(* IEC 61131-3 sources: volt/packages/volt-lsp-iec/test-corpus/lenze-mid/Device/Plc Logic/Application/Library Manager/CDSV3ProtocolUtils, 39 files *)

(* ---- PROTOCOLDATAUNIT.dut ---- *)
TYPE PROTOCOLDATAUNIT :
STRUCT
	PDATA : POINTER TO BYTE;
	DWSIZE : DWORD;
END_STRUCT
END_TYPE

(* ---- SERVICEHEADER.dut ---- *)
TYPE SERVICEHEADER :
STRUCT
	HEADERTAG : UINT := Constants.HeaderTagStandard;
	HEADERSIZE : UINT := UDINT_TO_UINT((SIZEOF(THIS^) - 4));
	SERVICEGROUP : UINT;
	SERVICE : UINT;
	DEVICESESSIONID : UDINT;
	SERVICELENGTH : UDINT;
	CUSTOMERID : UINT := 0;
	RESERVED : UINT := 0;
END_STRUCT
END_TYPE

(* ---- CONSTANTS.gvl ---- *)
VAR_GLOBAL
	HEADERTAGSTANDARD : UINT := 16#CD55;
	TAG_GENERALERROR : UINT := 16#FF7F;
	TAG_EXTENDEDERRORINFO : UINT := 16#FF7E;
END_VAR

(* ---- ERRORS.gvl ---- *)
VAR_GLOBAL
	ERR_PLCS_UNKNOWN_PROTOCOL : UDINT := 16#1011;
	ERR_PLCS_ALIGNMENT : UDINT := 16#1010;
	ERR_TSW_NOTCREATED : UDINT := 16#1000;
	ERR_TSR_NOMORETAGS : UDINT := 16#1040;
	ERR_TSR_NOCONTAINERTAG : UDINT := 16#1041;
	ERR_TSR_NODATATAG : UDINT := 16#1042;
	ERR_TSR_ENDOFTAG : UDINT := 16#1043;
	ERR_TSR_READONWRONGTAG : UDINT := 16#1044;
	ERR_TSR_NOTCREATED : UDINT := 16#1045;
END_VAR

(* ---- ICDSV3REQUESTBUILDER.itf ---- *)
INTERFACE ICDSV3REQUESTBUILDER
END_INTERFACE

METHOD BUILDREQUEST : UDINT
VAR_INPUT
	ITFSERVICEWRITER : IServiceWriter;
	XHASTOSWAP : BOOL;
END_VAR
END_METHOD

METHOD GETDATABUFFER : POINTER TO BYTE
END_METHOD

METHOD GETDATABUFFERSIZE : UDINT
END_METHOD

METHOD GETSERVICE : UINT
END_METHOD

METHOD GETSERVICEGROUP : UINT
END_METHOD

METHOD REQUESTENQUEUED : UDINT
END_METHOD

(* ---- ICDSV3REQUESTCALLBACK.itf ---- *)
INTERFACE ICDSV3REQUESTCALLBACK
END_INTERFACE

METHOD SETTARGETBYTEORDER
VAR_INPUT
	EBYTEORDER : IDatasources.ByteOrder;
END_VAR
END_METHOD

(* ---- IREQUESTRESULT.itf ---- *)
INTERFACE IREQUESTRESULT
END_INTERFACE

METHOD ISREPLYPENDING : BOOL
END_METHOD

METHOD SETREPLYPENDING
VAR_INPUT
	XREPLYPENDING : BOOL;
END_VAR
END_METHOD

(* ---- ISERVICEREADER.itf ---- *)
INTERFACE ISERVICEREADER
END_INTERFACE

METHOD GETCONTENT : UDINT
VAR_OUTPUT
	PDATA : POINTER TO BYTE;
END_VAR
END_METHOD

METHOD GETCONTENTSIZE : UDINT
VAR_OUTPUT
	CONTENTSIZE : UDINT;
END_VAR
END_METHOD

METHOD GETUNREADCONTENT : UDINT
VAR_OUTPUT
	PDATA : POINTER TO BYTE;
END_VAR
END_METHOD

METHOD GETUNREADCONTENTSIZE : UDINT
VAR_OUTPUT
	CONTENTSIZE : UDINT;
END_VAR
END_METHOD

METHOD IGNOREBYTES : UDINT
VAR_INPUT
	UDICOUNT : UDINT;
END_VAR
END_METHOD

METHOD MOVEDOWN : UDINT
END_METHOD

METHOD MOVENEXT : UDINT
END_METHOD

METHOD MOVENEXTCONDITIONAL : UDINT
VAR_INPUT
	BDOMOVE : BOOL;
END_VAR
END_METHOD

METHOD MOVEUP : UDINT
END_METHOD

METHOD READBYTE : UDINT
VAR_OUTPUT
	BT : BYTE;
END_VAR
END_METHOD

METHOD READBYTES : UDINT
VAR_INPUT
	PBUFFER : POINTER TO BYTE;
	UDICOUNT : UDINT;
END_VAR
END_METHOD

METHOD READBYTESSWAPPED : UDINT
VAR_INPUT
	PBUFFER : POINTER TO BYTE;
	UDICOUNT : UDINT;
END_VAR
END_METHOD

METHOD READDWORD : UDINT
VAR_OUTPUT
	DW : DWORD;
END_VAR
END_METHOD

METHOD READLWORD : UDINT
VAR_OUTPUT
	LW : LWORD;
END_VAR
END_METHOD

METHOD READSTRING : UDINT
VAR_OUTPUT
	STR : STRING(255);
END_VAR
END_METHOD

METHOD READWSTRING : UDINT
VAR_OUTPUT
	WSTR : WSTRING(255);
END_VAR
END_METHOD

METHOD READWORD : UDINT
VAR_OUTPUT
	WD : WORD;
END_VAR
END_METHOD

(* ---- ISERVICEWRITER.itf ---- *)
INTERFACE ISERVICEWRITER
END_INTERFACE

METHOD APPENDRAW : UDINT
VAR_INPUT
	PPDATA : POINTER TO POINTER TO BYTE;
	UDISIZE : UDINT;
END_VAR
END_METHOD

METHOD WRITEBYTE : UDINT
VAR_INPUT
	BT : BYTE;
END_VAR
END_METHOD

METHOD WRITEBYTES : UDINT
VAR_INPUT
	PDATA : POINTER TO BYTE;
	UDISIZE : UDINT;
END_VAR
END_METHOD

METHOD WRITEBYTESSWAPPED : UDINT
VAR_INPUT
	PDATA : POINTER TO BYTE;
	UDISIZE : UDINT;
END_VAR
END_METHOD

METHOD WRITECOMPLEXSTARTTAG : UDINT
VAR_INPUT
	UDITAG : UDINT;
	UDIMINLENSIZE : UDINT;
END_VAR
END_METHOD

METHOD WRITEDWORD : UDINT
VAR_INPUT
	DW : DWORD;
END_VAR
END_METHOD

METHOD WRITEDWORDSWAPPED : UDINT
VAR_INPUT
	DW : DWORD;
	BSWAP : BOOL;
END_VAR
END_METHOD

METHOD WRITEDATASTARTTAG : UDINT
VAR_INPUT
	UDITAG : UDINT;
	ALIGNMENT : CmpBinTagUtilIec.BTagAlignment;
	UDIMINLENSIZE : UDINT;
END_VAR
END_METHOD

METHOD WRITEENDTAG : UDINT
VAR_INPUT
	UDITAG : UDINT;
END_VAR
END_METHOD

METHOD WRITEFILLBYTES : UDINT
VAR_INPUT
	ALIGNMENT : CmpBinTagUtilIec.BTagAlignment;
END_VAR
END_METHOD

METHOD WRITELWORD : UDINT
VAR_INPUT
	LW : LWORD;
END_VAR
END_METHOD

METHOD WRITELWORDSWAPPED : UDINT
VAR_INPUT
	LW : LWORD;
	BSWAP : BOOL;
END_VAR
END_METHOD

METHOD WRITEPSTRING : UDINT
VAR_INPUT
	PSTR : POINTER TO STRING;
	UDILEN : UDINT;
END_VAR
END_METHOD

METHOD WRITESTRING : UDINT
VAR_INPUT
	STR : STRING(255);
END_VAR
END_METHOD

METHOD WRITEWORD : UDINT
VAR_INPUT
	WD : WORD;
END_VAR
END_METHOD

METHOD WRITEWORDSWAPPED : UDINT
VAR_INPUT
	WD : WORD;
	BSWAP : BOOL;
END_VAR
END_METHOD

(* ---- BUILDANDENQUEUEV3REQUEST.pou ---- *)
FUNCTION BUILDANDENQUEUEV3REQUEST : UDINT
VAR_INPUT
	ITFDATASOURCE : IDatasources.IDatasource;
	ITFCDSV3REQUESTBUILDER : ICDSV3RequestBuilder;
	ITFREQUESTCALLBACK : IDatasources.ICustomRequestCallback;
END_VAR
VAR_OUTPUT
	EREMOTEBYTEORDER : IDatasources.ByteOrder;
	XHASTOSWAP : BOOL;
	ITFCDSV3REQUEST : IDatasources.ICDSV3Request;
END_VAR
END_FUNCTION

(* ---- SWAPDWORD.pou ---- *)
FUNCTION SWAPDWORD
VAR_IN_OUT
	DW : DWORD;
END_VAR
END_FUNCTION

(* ---- SWAPDWORDIF.pou ---- *)
FUNCTION SWAPDWORDIF : DWORD
VAR_INPUT
	DW : DWORD;
	BYTEORDER : IDatasources.ByteOrder;
END_VAR
END_FUNCTION

(* ---- SWAPLWORD.pou ---- *)
FUNCTION SWAPLWORD
VAR_IN_OUT
	LW : LWORD;
END_VAR
END_FUNCTION

(* ---- SWAPWORD.pou ---- *)
FUNCTION SWAPWORD
VAR_IN_OUT
	WD : WORD;
END_VAR
END_FUNCTION

(* ---- SWAPWORDIF.pou ---- *)
FUNCTION SWAPWORDIF : WORD
VAR_INPUT
	W : WORD;
	BYTEORDER : IDatasources.ByteOrder;
END_VAR
END_FUNCTION

(* ---- UTILCHECKNATURALLYALIGNEDPOINTER.pou ---- *)
FUNCTION UTILCHECKNATURALLYALIGNEDPOINTER : UDINT
VAR_INPUT
	PTR : POINTER TO BYTE;
END_VAR
END_FUNCTION

(* ---- UTILGETLOCALBYTEORDER.pou ---- *)
FUNCTION UTILGETLOCALBYTEORDER : IDatasources.ByteOrder
END_FUNCTION

(* ---- UTILGETLOCALBYTEORDERATRUNTIME.pou ---- *)
FUNCTION UTILGETLOCALBYTEORDERATRUNTIME : IDatasources.ByteOrder
END_FUNCTION

(* ---- UTILHAVETOSWAPFORBINTAGUTIL.pou ---- *)
FUNCTION UTILHAVETOSWAPFORBINTAGUTIL : DINT
VAR_INPUT
	TARGETBYTEORDER : IDatasources.ByteOrder;
END_VAR
END_FUNCTION

(* ---- UTILISGENERALERRORREPLY.pou ---- *)
FUNCTION UTILISGENERALERRORREPLY : BOOL
VAR_INPUT
	PDU : ProtocolDataUnit;
	TARGETBYTEORDER : IDatasources.ByteOrder;
END_VAR
VAR_OUTPUT
	ERRORCODE : UDINT;
	RETRYTIME : UDINT;
END_VAR
END_FUNCTION

(* ---- UTILISINTELBYTEORDER.pou ---- *)
FUNCTION UTILISINTELBYTEORDER : BOOL
VAR_INPUT
	BO : IDatasources.ByteOrder;
END_VAR
END_FUNCTION

(* ---- UTILISTOSWAP.pou ---- *)
FUNCTION UTILISTOSWAP : BOOL
VAR_INPUT
	BO : IDatasources.ByteOrder;
END_VAR
END_FUNCTION

(* ---- UTILREADMISALIGNEDDWORD.pou ---- *)
FUNCTION UTILREADMISALIGNEDDWORD : DWORD
VAR_INPUT
	PDATA : POINTER TO BYTE;
	BO : IDatasources.ByteOrder;
END_VAR
END_FUNCTION

(* ---- UTILREADMISALIGNEDLWORD.pou ---- *)
FUNCTION UTILREADMISALIGNEDLWORD : LWORD
VAR_INPUT
	PDATA : POINTER TO BYTE;
	BO : IDatasources.ByteOrder;
END_VAR
END_FUNCTION

(* ---- UTILREADMISALIGNEDWORD.pou ---- *)
FUNCTION UTILREADMISALIGNEDWORD : WORD
VAR_INPUT
	PDATA : POINTER TO BYTE;
	BO : IDatasources.ByteOrder;
END_VAR
END_FUNCTION

(* ---- UTILSWRITEBYTE.pou ---- *)
FUNCTION UTILSWRITEBYTE : UDINT
VAR_INPUT
	ITFSERVICEWRITER : IServiceWriter;
	UITAG : UINT;
	BYVALUE : BYTE;
END_VAR
END_FUNCTION

(* ---- UTILSWRITESTRING.pou ---- *)
FUNCTION UTILSWRITESTRING : UDINT
VAR_INPUT
	ITFWRITER : IServiceWriter;
	UITAG : UINT;
	PSZ : POINTER TO STRING(255);
END_VAR
END_FUNCTION

(* ---- UTILSWRITEUDINT.pou ---- *)
FUNCTION UTILSWRITEUDINT : UDINT
VAR_INPUT
	ITFSERVICEWRITER : IServiceWriter;
	UITAG : UINT;
	UDIVALUE : UDINT;
	XHASTOSWAP : BOOL;
END_VAR
END_FUNCTION

(* ---- UTILSWRITEUINT.pou ---- *)
FUNCTION UTILSWRITEUINT : UDINT
VAR_INPUT
	ITFSERVICEWRITER : IServiceWriter;
	UITAG : UINT;
	UIVALUE : UINT;
	XHASTOSWAP : BOOL;
END_VAR
END_FUNCTION

(* ---- UTILSWRITEULINT.pou ---- *)
FUNCTION UTILSWRITEULINT : UDINT
VAR_INPUT
	ITFSERVICEWRITER : IServiceWriter;
	UITAG : UINT;
	ULIVALUE : ULINT;
	XHASTOSWAP : BOOL;
END_VAR
END_FUNCTION

(* ---- UTILVALIDATEBYTEORDER.pou ---- *)
FUNCTION UTILVALIDATEBYTEORDER : BOOL
VAR_IN_OUT
	BO : IDatasources.Byteorder;
END_VAR
END_FUNCTION

(* ---- DEFAULTREQUESTRESULT.pou ---- *)
FUNCTION_BLOCK DEFAULTREQUESTRESULT
VAR
	M_XREPLYPENDING : BOOL;
END_VAR
END_FUNCTION_BLOCK

METHOD ISREPLYPENDING : BOOL
END_METHOD

METHOD SETREPLYPENDING
VAR_INPUT
	XREPLYPENDING : BOOL;
END_VAR
END_METHOD

(* ---- SERVICEREADER.pou ---- *)
FUNCTION_BLOCK SERVICEREADER
VAR
	_HBTR : CmpBinTagUtilIec.RTS_IEC_HANDLE := CmpBinTagUtilIec.RTS_INVALID_HANDLE;
	_PCURRENTCONTENT : POINTER TO BYTE;
	_UDICURRENTCONTENTLENGTH : UDINT;
	_UDIPOSITION : UDINT;
	_CURRENTTAGTYPE : CmpBinTagUtilIec.BTagElementType;
	_TARGETBYTEORDER : IDatasources.ByteOrder;
	ALIVE : BOOL;
	ISDATATAG : BOOL;
	PRVTOPLEVEL : BOOL;
	TAGID : UDINT;
	VALIDTAG : BOOL;
END_VAR
END_FUNCTION_BLOCK

METHOD CREATE : UDINT
VAR_INPUT
	PREADERBUFFER : POINTER TO BYTE;
	UDIREADERBUFFERSIZE : UDINT;
	PDATABUFFER : POINTER TO BYTE;
	UDIDATABUFFERSIZE : UDINT;
	TARGETBYTEORDER : IDatasources.ByteOrder;
END_VAR
END_METHOD

METHOD CREATEDYNAMIC : UDINT
VAR_INPUT
	PDATABUFFER : POINTER TO BYTE;
	UDIDATABUFFERSIZE : UDINT;
	TARGETBYTEORDER : IDatasources.ByteOrder;
END_VAR
END_METHOD

METHOD DESTROY : UDINT
END_METHOD

METHOD FB_EXIT : BOOL
VAR_INPUT
	BINCOPYCODE : BOOL;
END_VAR
END_METHOD

METHOD GETCONTENT : UDINT
VAR_OUTPUT
	PDATA : POINTER TO BYTE;
END_VAR
END_METHOD

METHOD GETCONTENTSIZE : UDINT
VAR_OUTPUT
	CONTENTSIZE : UDINT;
END_VAR
END_METHOD

METHOD GETUNREADCONTENT : UDINT
VAR_OUTPUT
	PDATA : POINTER TO BYTE;
END_VAR
END_METHOD

METHOD GETUNREADCONTENTSIZE : UDINT
VAR_OUTPUT
	CONTENTSIZE : UDINT;
END_VAR
END_METHOD

METHOD IGNOREBYTES : UDINT
VAR_INPUT
	UDICOUNT : UDINT;
END_VAR
END_METHOD

METHOD MOVEDOWN : UDINT
END_METHOD

METHOD MOVENEXT : UDINT
END_METHOD

METHOD MOVENEXTCONDITIONAL : UDINT
VAR_INPUT
	BDOMOVE : BOOL;
END_VAR
END_METHOD

METHOD MOVEUP : UDINT
END_METHOD

METHOD READBYTE : UDINT
VAR_OUTPUT
	BT : BYTE;
END_VAR
END_METHOD

METHOD READBYTES : UDINT
VAR_INPUT
	PBUFFER : POINTER TO BYTE;
	UDICOUNT : UDINT;
END_VAR
END_METHOD

METHOD READBYTESSWAPPED : UDINT
VAR_INPUT
	PBUFFER : POINTER TO BYTE;
	UDICOUNT : UDINT;
END_VAR
END_METHOD

METHOD READDWORD : UDINT
VAR_OUTPUT
	DW : DWORD;
END_VAR
END_METHOD

METHOD READLWORD : UDINT
VAR_OUTPUT
	LW : LWORD;
END_VAR
END_METHOD

METHOD READSTRING : UDINT
VAR_OUTPUT
	STR : STRING(255);
END_VAR
END_METHOD

METHOD READWSTRING : UDINT
VAR_OUTPUT
	WSTR : WSTRING(255);
END_VAR
END_METHOD

METHOD READWORD : UDINT
VAR_OUTPUT
	WD : WORD;
END_VAR
END_METHOD

METHOD PRVINIT : UDINT
VAR_INPUT
	PDATABUFFER : POINTER TO BYTE;
	UDIDATABUFFERSIZE : UDINT;
END_VAR
END_METHOD

METHOD PRVREADSTARTTAG : UDINT
END_METHOD

(* ---- SERVICEREQUEST.pou ---- *)
FUNCTION_BLOCK SERVICEREQUEST EXTENDS ServiceRequestBase
VAR
	_WRITER : ServiceWriter;
	_HSAVEPOINT : CmpBinTagUtilIec.RTS_IEC_HANDLE := CmpBinTagUtilIec.RTS_INVALID_HANDLE;
	WRITER : IServiceWriter;
END_VAR
END_FUNCTION_BLOCK

METHOD CREATE : UDINT
VAR_INPUT
	TARGETBYTEORDER : IDatasources.ByteOrder;
	UISERVICEGROUP : UINT;
	UISERVICE : UINT;
	UDIDEVSESSID : UDINT;
	PBUFFER : POINTER TO BYTE;
	UDIBUFFERSIZE : UDINT;
END_VAR
END_METHOD

METHOD FB_EXIT : BOOL
VAR_INPUT
	BINCOPYCODE : BOOL;
END_VAR
END_METHOD

METHOD RESTORESAVEPOINT : UDINT
END_METHOD

METHOD STORESAVEPOINT : UDINT
END_METHOD

METHOD DOFINISH : UDINT
VAR_INPUT
	XDESTROYONLY : BOOL;
END_VAR
VAR_OUTPUT
	PDUCONTENT : ProtocolDataUnit;
END_VAR
END_METHOD

METHOD PRVDISPOSE : UDINT
END_METHOD

METHOD PRVFREESAVEPOINT : BOOL
END_METHOD

(* ---- SERVICEREQUESTBASE.pou ---- *)
FUNCTION_BLOCK SERVICEREQUESTBASE
VAR
	_PHEADER : POINTER TO ServiceHeader;
	_PDU : ProtocolDataUnit;
	_BPDUVALID : BOOL;
	_BO : IDatasources.ByteOrder;
	_BSWAP : BOOL;
	_UDIMAXCONTENTSIZE : UDINT;
	HEADERSIZE : UDINT := SIZEOF(_pHeader^);
	CONTENTPTR : POINTER TO BYTE;
	DATA : ProtocolDataUnit;
	DATAVALID : BOOL;
	HAVETOSWAP : BOOL;
	HEADER : ServiceHeader;
END_VAR
END_FUNCTION_BLOCK

METHOD CREATE : UDINT
VAR_INPUT
	TARGETBYTEORDER : IDatasources.ByteOrder;
	UISERVICEGROUP : UINT;
	UISERVICE : UINT;
	UDIDEVSESSID : UDINT;
	PBUFFER : POINTER TO BYTE;
	UDIBUFFERSIZE : UDINT;
END_VAR
END_METHOD

METHOD FB_EXIT : BOOL
VAR_INPUT
	BINCOPYCODE : BOOL;
END_VAR
END_METHOD

METHOD FINISH : UDINT
VAR_INPUT
	BDESTROYONLY : BOOL;
END_VAR
END_METHOD

METHOD DOFINISH : UDINT
VAR_INPUT
	XDESTROYONLY : BOOL;
END_VAR
VAR_OUTPUT
	PDUCONTENT : ProtocolDataUnit;
END_VAR
END_METHOD

METHOD PRVSWAPHEADER : UDINT
END_METHOD

(* ---- SERVICEREQUESTRAW.pou ---- *)
FUNCTION_BLOCK SERVICEREQUESTRAW EXTENDS ServiceRequestBase
VAR
	_PDURAW : ProtocolDataUnit;
	RAWDATA : ProtocolDataUnit;
END_VAR
END_FUNCTION_BLOCK

METHOD DOFINISH : UDINT
VAR_INPUT
	XDESTROYONLY : BOOL;
END_VAR
VAR_OUTPUT
	PDUCONTENT : ProtocolDataUnit;
END_VAR
END_METHOD

(* ---- SERVICERESPONSE.pou ---- *)
FUNCTION_BLOCK SERVICERESPONSE
VAR
	_HEADERCOPY : ServiceHeader;
	_PDATA : POINTER TO BYTE;
	_BO : IDatasources.ByteOrder;
	_READER : ServiceReader;
	_PBYCONTENTDATA : POINTER TO BYTE;
	_UXICONTENTSIZE : __UXINT;
	CONTENTDATA : POINTER TO BYTE;
	CONTENTSIZE : __UXINT;
	HEADER : ServiceHeader;
	READER : IServiceReader;
END_VAR
END_FUNCTION_BLOCK

METHOD CREATE : UDINT
VAR_INPUT
	PDATA : POINTER TO BYTE;
	DWSIZE : DWORD;
	TARGETBYTEORDER : IDatasources.ByteOrder;
	UIHEADERTAG : UINT;
END_VAR
END_METHOD

METHOD CREATEPDU : UDINT
VAR_INPUT
	PDU : ProtocolDataUnit;
	TARGETBYTEORDER : IDatasources.ByteOrder;
	UIHEADERTAG : UINT;
END_VAR
END_METHOD

METHOD DESTROY : UDINT
END_METHOD

METHOD FB_EXIT : BOOL
VAR_INPUT
	BINCOPYCODE : BOOL;
END_VAR
END_METHOD

METHOD PRVANALYZEHEADEROBSOLETE : UDINT
VAR_INPUT
	PDATA : POINTER TO BYTE;
	DWSIZE : DWORD;
	TARGETBYTEORDER : IDatasources.ByteOrder;
	UIHEADERTAG : UINT;
END_VAR
END_METHOD

METHOD PRVCOPYHEADER : UDINT
VAR_INPUT
	PHEADER : POINTER TO ServiceHeader;
END_VAR
END_METHOD

METHOD PRVDISPOSE : UDINT
END_METHOD

(* ---- SERVICEWRITER.pou ---- *)
FUNCTION_BLOCK SERVICEWRITER
VAR
	_HBTW : CmpBinTagUtilIec.RTS_IEC_HANDLE := CmpBinTagUtilIec.RTS_INVALID_HANDLE;
	ALIVE : BOOL;
	HANDLE : CmpBinTagUtilIec.RTS_IEC_HANDLE;
END_VAR
END_FUNCTION_BLOCK

METHOD CREATE : UDINT
VAR_INPUT
	PWRITERBUFFER : POINTER TO BYTE;
	UDIWRITERBUFFERSIZE : UDINT;
	PDATABUFFER : POINTER TO BYTE;
	UDIDATABUFFERSIZE : UDINT;
	TARGETBYTEORDER : IDatasources.ByteOrder;
END_VAR
END_METHOD

METHOD CREATEDYNAMIC : UDINT
VAR_INPUT
	PDATABUFFER : POINTER TO BYTE;
	UDIDATABUFFERSIZE : UDINT;
	TARGETBYTEORDER : IDatasources.ByteOrder;
END_VAR
END_METHOD

METHOD DESTROY : UDINT
END_METHOD

METHOD FB_EXIT : BOOL
VAR_INPUT
	BINCOPYCODE : BOOL;
END_VAR
END_METHOD

METHOD FINISH : UDINT
VAR_IN_OUT
	PWRITTENDATA : POINTER TO BYTE;
	UDIWRITTENSIZE : UDINT;
END_VAR
END_METHOD

METHOD APPENDRAW : UDINT
VAR_INPUT
	PPDATA : POINTER TO POINTER TO BYTE;
	UDISIZE : UDINT;
END_VAR
END_METHOD

METHOD WRITEBYTE : UDINT
VAR_INPUT
	BT : BYTE;
END_VAR
END_METHOD

METHOD WRITEBYTES : UDINT
VAR_INPUT
	PDATA : POINTER TO BYTE;
	UDISIZE : UDINT;
END_VAR
END_METHOD

METHOD WRITEBYTESSWAPPED : UDINT
VAR_INPUT
	PDATA : POINTER TO BYTE;
	UDISIZE : UDINT;
END_VAR
END_METHOD

METHOD WRITECOMPLEXSTARTTAG : UDINT
VAR_INPUT
	UDITAG : UDINT;
	UDIMINLENSIZE : UDINT;
END_VAR
END_METHOD

METHOD WRITEDWORD : UDINT
VAR_INPUT
	DW : DWORD;
END_VAR
END_METHOD

METHOD WRITEDWORDSWAPPED : UDINT
VAR_INPUT
	DW : DWORD;
	BSWAP : BOOL;
END_VAR
END_METHOD

METHOD WRITEDATASTARTTAG : UDINT
VAR_INPUT
	UDITAG : UDINT;
	ALIGNMENT : CmpBinTagUtilIec.BTagAlignment;
	UDIMINLENSIZE : UDINT;
END_VAR
END_METHOD

METHOD WRITEENDTAG : UDINT
VAR_INPUT
	UDITAG : UDINT;
END_VAR
END_METHOD

METHOD WRITEFILLBYTES : UDINT
VAR_INPUT
	ALIGNMENT : CmpBinTagUtilIec.BTagAlignment;
END_VAR
END_METHOD

METHOD WRITELWORD : UDINT
VAR_INPUT
	LW : LWORD;
END_VAR
END_METHOD

METHOD WRITELWORDSWAPPED : UDINT
VAR_INPUT
	LW : LWORD;
	BSWAP : BOOL;
END_VAR
END_METHOD

METHOD WRITEPSTRING : UDINT
VAR_INPUT
	PSTR : POINTER TO STRING;
	UDILEN : UDINT;
END_VAR
END_METHOD

METHOD WRITESTRING : UDINT
VAR_INPUT
	STR : STRING(255);
END_VAR
END_METHOD

METHOD WRITEWORD : UDINT
VAR_INPUT
	WD : WORD;
END_VAR
END_METHOD

METHOD WRITEWORDSWAPPED : UDINT
VAR_INPUT
	WD : WORD;
	BSWAP : BOOL;
END_VAR
END_METHOD

METHOD PRVINIT : UDINT
VAR_INPUT
	PDATABUFFER : POINTER TO BYTE;
	UDIDATABUFFERSIZE : UDINT;
	TARGETBYTEORDER : IDatasources.ByteOrder;
END_VAR
END_METHOD

(* ---- SERVICEWRITERSAVEPOINT.pou ---- *)
FUNCTION_BLOCK SERVICEWRITERSAVEPOINT
VAR
	_HWRITER : CmpBinTagUtilIec.RTS_IEC_HANDLE;
	_HSAVEPOINT : CmpBinTagUtilIec.RTS_IEC_HANDLE := CmpBinTagUtilIec.RTS_INVALID_HANDLE;
	_DATA : ARRAY [0..500] OF DWORD;
END_VAR
END_FUNCTION_BLOCK

METHOD FB_EXIT : BOOL
VAR_INPUT
	BINCOPYCODE : BOOL;
END_VAR
END_METHOD

METHOD FREESAVEPOINT : UDINT
END_METHOD

METHOD INIT : UDINT
VAR_IN_OUT
	WRITER : ServiceWriter;
END_VAR
END_METHOD

METHOD RESTORE : UDINT
END_METHOD

METHOD STORE : UDINT
END_METHOD
